{attribute 'linkalways'} 
{attribute 'no_explicit_call' := 'This FB is a CLASS and must be accessed using methods or properties'}
{attribute 'enable_dynamic_creation'}
FUNCTION_BLOCK _ULINT EXTENDS NumericDatatypeBase
VAR
	localData : ULINT;
	activeData : REFERENCE TO ULINT REF= localData;
END_VAR

PROPERTY PUBLIC Address : PVOID
GET
Address := ADR(activeData);
END_GET
END_PROPERTY

METHOD PUBLIC ClearReference
VAR_INPUT
END_VAR
activeData REF= localData;
END_METHOD

METHOD PUBLIC Clone : I_Datatype
VAR
    pClone : POINTER TO _ULINT;
END_VAR
pClone := __NEW(_ULINT(InitialValue := Value));
Clone := pClone^;
END_METHOD

METHOD FB_init : BOOL
VAR_INPUT
	bInitRetains : BOOL; // if TRUE, the retain variables are initialized (warm start / cold start)
	bInCopyCode : BOOL;  // if TRUE, the instance afterwards gets moved into the copy code (online change)
	InitialValue : ULINT;
END_VAR
localData := InitialValue;
END_METHOD

PROPERTY PUBLIC IsFloat : BOOL
GET
IsFloat := FALSE;
END_GET
END_PROPERTY

PROPERTY PUBLIC IsSigned : BOOL
GET
IsSigned := FALSE;
END_GET
END_PROPERTY

METHOD PUBLIC MakeReferenceTo
VAR_INPUT
	ReferenceTarget : REFERENCE TO ULINT;
END_VAR
activeData REF= ReferenceTarget;
END_METHOD

PROPERTY PUBLIC MaxValue : ULINT
GET
MaxValue :=  DatatypeLimits.ULINT_MAX_VALUE;
END_GET
END_PROPERTY

PROPERTY PUBLIC MinValue : ULINT
GET
MinValue := DatatypeLimits.ULINT_MIN_VALUE;
END_GET
END_PROPERTY

METHOD PROTECTED SerializeMaxValue
VAR_INPUT
	Serializer : I_Serializer;
END_VAR
Serializer.AddUlint(MaxValue);
END_METHOD

METHOD PROTECTED SerializeMinValue
VAR_INPUT
	Serializer : I_Serializer;
END_VAR
Serializer.AddUlint(MinValue);
END_METHOD

METHOD PUBLIC SerializeWith
VAR_INPUT
	Serializer : I_Serializer;
END_VAR
Serializer.AddUlint(activeData);
END_METHOD

PROPERTY PUBLIC Size : UDINT
GET
Size := SIZEOF(activeData);
END_GET
END_PROPERTY

METHOD TryDeserializeFrom : BOOL
VAR_INPUT
	Deserializer : I_Deserializer;
	Feedback : I_DeserializerFeedback;
END_VAR
TryDeserializeFrom := Deserializer.TryGetUlint(activeData, Feedback);
END_METHOD

METHOD TryMakeReferenceTo : BOOL
VAR_INPUT
	Target : I_Datatype;
END_VAR
VAR
	pTargetData : POINTER TO ULINT;
END_VAR
IF NOT (Target.TypeName = TypeName) THEN
	RETURN;
END_IF

pTargetData := Target.Address;
activeData REF= pTargetData^;
TryMakeReferenceTo := TRUE;
END_METHOD

PROPERTY PUBLIC TypeName : T_MAXSTRING
GET
TypeName := 'ULINT';
END_GET
END_PROPERTY

PROPERTY PUBLIC Value : REFERENCE TO ULINT
GET
Value REF= activeData;
END_GET
END_PROPERTY

END_FUNCTION_BLOCK

(* stored: Version 1.1.0.1, ProductVersion 3.1.4024.12
   POU _ULINT: Id {15620a13-49a3-49da-bc73-2e6e2b844d97}, SpecialFunc None
   Folder Constructor: Id {0fab894d-6fce-4f32-a82c-40e3d215bc46}
   Folder Protected: Id {ebd8af2b-8afe-4503-897f-977a527be49d}
   Property Address: Id {2a665eb0-ee93-45f1-8804-bdf0753fdfa5}
   Get Get: Id {18ccab72-2dff-4ffc-a0dc-738702eecfb4}
   Method ClearReference: Id {e93a83af-5ce9-42fb-a834-1a3a71adf17e}
   Method Clone: Id {6d98c70f-31c6-432b-8d75-713faf0c0c8f}
   Method FB_init: Id {f9bb6245-1776-4515-af79-3b41c29bf794}
   Property IsFloat: Id {52abe5a4-cf31-4e39-ba1e-dd4a3be46b64}
   Get Get: Id {8d1b1f3a-ecaf-449a-9f07-9828e2c51b82}
   Property IsSigned: Id {9e786c82-c1ad-45c3-bc98-471d6ecaba7d}
   Get Get: Id {555e5d28-7be1-4915-be06-6ab5f7246872}
   Method MakeReferenceTo: Id {bee8dc61-1a19-4f07-948c-7fc6f5d1649b}
   Property MaxValue: Id {401104ba-c18a-4cad-9693-4451a52c7e5e}
   Get Get: Id {6ebf1750-e3ec-467a-a82c-c35ac31a3ea9}
   Property MinValue: Id {a64f8e2a-1b2b-4414-8c21-dcca44bc392b}
   Get Get: Id {440f2586-a60a-4bbb-a78d-7e5e14af5818}
   Method SerializeMaxValue: Id {3d607e4d-d540-4370-857a-2ad54e412ed0}
   Method SerializeMinValue: Id {933b3da6-536a-4c5f-acc6-03e5fffba51f}
   Method SerializeWith: Id {07d6c5d4-1307-407e-a05f-7c8ca221ed13}
   Property Size: Id {60844251-ed2d-4c77-88e6-0671ffe0d444}
   Get Get: Id {2e98d5e3-f26a-4696-93c4-8e89b4bfdcac}
   Method TryDeserializeFrom: Id {69ee5c4f-587e-4333-adb2-b07e12275911}
   Method TryMakeReferenceTo: Id {56720a69-3925-4547-bb48-419cd11c9f58}
   Property TypeName: Id {55403037-d8c2-4b0f-861f-64a66c64e6d2}
   Get Get: Id {4d283c5e-843b-444a-8ff6-fc6d105a59b3}
   Property Value: Id {70b16337-af33-4ec6-9b65-9e82b4f427a4}
   Get Get: Id {6b034a19-1fb8-4685-a2ae-fbeb93531182} *)
